FUNCTION_BLOCK BOOL_Param
VAR_INPUT PERSISTENT
	val				: BOOL;
END_VAR

END_FUNCTION_BLOCK

(* stored: Version 1.1.0.1
   POU BOOL_Param: Id {9856de7c-b804-4e12-856d-47a6d6134cf1}, SpecialFunc None *)
